// TwinCAT 3 PLC project tcl_TwinCAT_UnitTestLibrary_Learning_Space
// ProgramVersion: 3.1.4024.0
// libraries:
//   Tc2_Standard, * (Beckhoff Automation GmbH)
//   Tc2_System, * (Beckhoff Automation GmbH)
//   Tc3_Module, * (Beckhoff Automation GmbH)
//   tcl_UnitTestLibrary, * (Red Rock Controls Limited)
// project tree:
//   Classes/ MyCalculatorClass.TcPOU
//   / PlcTask.TcTTO
//   POUs/ MAIN.TcPOU
//   TestSuites/ MyCalculatorTestSuite.TcPOU
//   Tests/ DivideByTwoTest.TcPOU, DivideByZeroTest.TcPOU
// (motion and I/O tree: see PLC project tcunit_learning_space)
// real-time tasks:
//   TASK PlcTask: cycle T#10ms, priority 20, ADS port 350
//   TASK PlcTask1: cycle T#10ms, priority 21, ADS port 351
//   TASK PlcTask2: cycle T#10ms, priority 22, ADS port 352

CONFIGURATION tcl_TwinCAT_UnitTestLibrary_Learning_Space
    RESOURCE PLC ON TwinCAT3
        TASK PlcTask(INTERVAL := T#10ms, PRIORITY := 22);
        PROGRAM MAIN WITH PlcTask : MAIN;
    END_RESOURCE
END_CONFIGURATION

// ---- POUs/MAIN.TcPOU
PROGRAM MAIN
VAR
	CalcTestSuite : MyCalculatorTestSuite;
END_VAR

CalcTestSuite();

END_PROGRAM

// ---- TestSuites/MyCalculatorTestSuite.TcPOU
FUNCTION_BLOCK MyCalculatorTestSuite
VAR
	_DivideByZeroTest : DivideByZeroTest;
	_DivideByTwoTest : DivideByTwoTest;
END_VAR

_DivideByZeroTest.RunTest();
_DivideByTwoTest.RunTest();

END_FUNCTION_BLOCK

// ---- Tests/DivideByZeroTest.TcPOU
FUNCTION_BLOCK DivideByZeroTest EXTENDS T_UnitTestBase
VAR
	myCalculator : MyCalculatorClass;
END_VAR

{attribute 'analysis' := '-33'} // inhibit unused variable warning
METHOD  RunTest
TestCompleted := AssertEquals_INT(Expected := -1,
						Actual := myCalculator.Divide(2,0),
						Message := 'Calculator did not reject a divide by zero');
END_METHOD

END_FUNCTION_BLOCK

// ---- Classes/MyCalculatorClass.TcPOU
FUNCTION_BLOCK MyCalculatorClass
VAR
END_VAR

METHOD Divide : INT
VAR_INPUT
	x : INT;
	y : INT;
END_VAR
IF y <> 0 THEN
	Divide := x/y;
ELSE
	Divide := -1;
END_IF
END_METHOD

END_FUNCTION_BLOCK

// ---- Tests/DivideByTwoTest.TcPOU
FUNCTION_BLOCK DivideByTwoTest EXTENDS T_UnitTestBase
VAR
	myCalculator : MyCalculatorClass;
END_VAR

{attribute 'analysis' := '-33'} // inhibit unused variable warning
METHOD  RunTest
IF NOT TestCompleted THEN
	 AssertEquals_INT(Expected := 1,
						Actual := myCalculator.Divide(2,2),
						Message := 'Calculator failed correct division by two');
END_IF
END_METHOD

END_FUNCTION_BLOCK
